FUNCTION_BLOCK Q_ChangePolygonPoint (* Command Change Polygon Point( Part 6 - F.52 ) *)
  (* Standard: ISO 11783-6; Description: This command is used by a Working Set to modify a point in an Output Polygon object. Return values iso_s16 - E_NO_ERR - OK - E_OVERFLOW - buffer overflow - E_NOACT - Command not possible in current state - E_NO_INSTANCE - No VT client available *)
  (* Version 1.0, 2022-07-08, franz *)
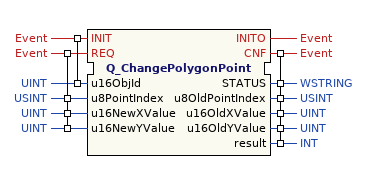
  EVENT_INPUT
    INIT WITH u16ObjId; (* Service Initialization *)
    REQ WITH u8PointIndex, u16NewXValue, u16NewYValue; (* Service Request *)
  END_EVENT
  EVENT_OUTPUT
    INITO; (* Initialization Confirm *)
    CNF WITH STATUS, result, u8OldPointIndex, u16OldXValue, u16OldYValue; (* Confirmation of Requested Service *)
  END_EVENT
  VAR_INPUT
    u16ObjId : UINT; (* Object ID of the Output Polygon object to change *)
    u8PointIndex : USINT; (* Point index of the point to replace. *)
    u16NewXValue : UINT; (* New X value of a point relative to the top left corner of the polygon *)
    u16NewYValue : UINT; (* New Y value of a point relative to the top left corner of the polygon *)
  END_VAR
  VAR_OUTPUT
    STATUS : WSTRING; (* Service Status *)
    u8OldPointIndex : USINT; (* Old point index of the point to replace. *)
    u16OldXValue : UINT; (* Old X value of a point relative to the top left corner of the polygon *)
    u16OldYValue : UINT; (* Old Y value of a point relative to the top left corner of the polygon *)
    result : INT; (* retval see description *)
  END_VAR
END_FUNCTION_BLOCK
